(* CODESYS project tcbase2.library
   Company: Beckhoff Automation GmbH
   Title: Tc2_Base2
   Placeholder: Tc2_Base2
   Version: 1.0.0.0

Project tree, tasks and I/O mapping:
  libraries: Tc2_System, * (Beckhoff Automation GmbH)
  Data types/
    data type FW_ULINT
  Global Variables/
    global variables Global_Variables
  POUs/
    function FW_GetActualDcTime2 [ST]
    function FW_GetCurDcTaskTime2 [ST]
    function FW_GetCurDcTickTime2 [ST]
    function FW_GetCurTaskSystemTime2 [ST]
  Visualizations/
*)

// Data types/FW_ULINT
TYPE FW_ULINT :
STRUCT
	loUDINT : UDINT;
	hiUDINT : UDINT;
END_STRUCT
END_TYPE

// Global Variables/Global_Variables
VAR_GLOBAL
END_VAR

// POUs/FW_GetActualDcTime2
FUNCTION FW_GetActualDcTime2 : UDINT
VAR_INPUT
	p: POINTER TO FW_ULINT;
END_VAR
VAR
END_VAR

;

END_FUNCTION

// POUs/FW_GetCurDcTaskTime2
FUNCTION FW_GetCurDcTaskTime2 : UDINT
VAR_INPUT
	p: POINTER TO FW_ULINT;
END_VAR
VAR
END_VAR

;

END_FUNCTION

// POUs/FW_GetCurDcTickTime2
FUNCTION FW_GetCurDcTickTime2 : UDINT
VAR_INPUT
	p: POINTER TO FW_ULINT;
END_VAR
VAR
END_VAR

;

END_FUNCTION

// POUs/FW_GetCurTaskSystemTime2
FUNCTION FW_GetCurTaskSystemTime2 : UDINT
VAR_INPUT
	p: POINTER TO FW_ULINT;
END_VAR
VAR
END_VAR

;

END_FUNCTION
